{attribute 'linkalways'} 
{attribute 'no_explicit_call' := 'This FB is a CLASS and must be accessed using methods or properties'}
{attribute 'enable_dynamic_creation'}
FUNCTION_BLOCK FINAL GT_LINT EXTENDS Node
VAR
	in1 : _LINT(0);
	in2 : _LINT(0);
	out : _BOOL(FALSE);
END_VAR

METHOD PUBLIC Clone : I_Node
VAR
	pNode : POINTER TO GT_LINT;
END_VAR
pNode := __NEW(GT_LINT);
Clone := pNode^;
END_METHOD

METHOD FB_init : BOOL
VAR_INPUT
	bInitRetains : BOOL; // if TRUE, the retain variables are initialized (warm start / cold start)
	bInCopyCode : BOOL;  // if TRUE, the instance afterwards gets moved into the copy code (online change)
END_VAR
AddInput('in1',THIS^.in1);
AddInput('in2',THIS^.in2);
AddOutput('out', THIS^.out);
END_METHOD

METHOD PROTECTED OnExecute
VAR
END_VAR
out.Value := in1.Value > in2.Value;
END_METHOD

END_FUNCTION_BLOCK

(* stored: Version 1.1.0.1, ProductVersion 3.1.4024.15
   POU GT_LINT: Id {ff93e1d0-86ef-46c2-b2df-5da48ee857eb}, SpecialFunc None
   Folder Constructor: Id {c6194c2c-6c3e-42e1-8a91-d58d559ff4e1}
   Method Clone: Id {1e252b1a-ae82-4ef2-978f-32212fabb741}
   Method FB_init: Id {d232d3b4-4c97-4c6e-957c-fb5415fe7d4d}
   Method OnExecute: Id {cb4e9c1a-da94-4230-ba73-07b8a7c59e99} *)
